FUNCTION_BLOCK BfbIDMTCurve
  (* Standard: 61499-2 *)
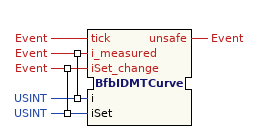
  EVENT_INPUT
    tick;
    i_measured WITH i;
    iSet_change WITH iSet;
  END_EVENT
  EVENT_OUTPUT
    unsafe;
  END_EVENT
  VAR_INPUT
    i : USINT;
    iSet : USINT;
  END_VAR
  VAR
    cnt : ULINT := 0;
    max : LREAL := 0;
    k : REAL := 100;
    b : REAL := 0.135;
    a : REAL := 1.0;
  END_VAR
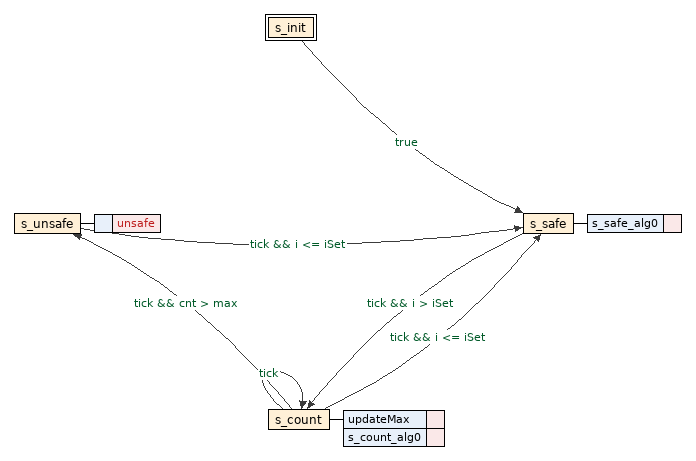
  EC_STATES
    s_init;
    s_safe : s_safe_alg0;
    s_count : updateMax, s_count_alg0;
    s_unsafe : -> unsafe;
  END_STATES
  EC_TRANSITIONS
    s_init TO s_safe := true;
    s_safe TO s_count := tick && i > iSet;
    s_count TO s_safe := tick && i <= iSet;
    s_count TO s_unsafe := tick && cnt > max;
    s_count TO s_count := tick;
    s_unsafe TO s_safe := tick && i <= iSet;
  END_TRANSITIONS
  ALGORITHM s_safe_alg0 IN ST:
cnt := 0;
  END_ALGORITHM
  ALGORITHM s_count_alg0 IN ST:
cnt := cnt + 1;
  END_ALGORITHM
  ALGORITHM updateMax IN C:
        me->max = ((me->k*me->b) / (pow((me->i / me->iSet),me->a) - 1));
  END_ALGORITHM
END_FUNCTION_BLOCK
